{attribute 'GeneratedUsingTerminal: IODEVICETYPE_ETHERCATPROT'}
{attribute addProperty BoxType "IODEVICETYPE_ETHERCATPROT"}
{attribute addProperty Id "Beckhoff_EM2xxxBeckhoff_EM2xxx_23EB33C640Beckhoff_EM3xxxBeckhoff_EM3xxx_ABA3179978Beckhoff_EM7xxxBeckhoff_EM7xxx_110CC3B3681SyncUnitsSyncUnits_99E584AF18InputsInputs_25A0042B160OutputsOutputs_2397A10E106InfoDataInfoData_E68C61CD28"}
{attribute addProperty CRC "1180849743"}
{attribute addProperty Size "1111"}
TYPE EtherCAT_Master_EMxxxx_4662564F :
STRUCT
	{attribute addProperty Name "Beckhoff_EM2xxx"}
	{attribute addProperty PreviousPort "EtherCAT_Master_EMxxxx : Master"}
	Beckhoff_EM2xxx : Beckhoff_EM2xxx_23EB33C6;
	{attribute addProperty Name "Beckhoff_EM3xxx"}
	{attribute addProperty PreviousPort "Beckhoff EM2xxx : C"}
	Beckhoff_EM3xxx : Beckhoff_EM3xxx_ABA31799;
	{attribute addProperty Name "Beckhoff_EM7xxx"}
	{attribute addProperty PreviousPort "Beckhoff EM3xxx : C"}
	Beckhoff_EM7xxx : Beckhoff_EM7xxx_110CC3B3;
	{attribute addProperty Name "SyncUnits"}
	SyncUnits : SyncUnits_99E584AF;
	{attribute addProperty Name "Inputs"}
	Inputs : Inputs_25A0042B;
	{attribute addProperty Name "Outputs"}
	Outputs : Outputs_2397A10E;
	{attribute addProperty Name "InfoData"}
	InfoData : InfoData_E68C61CD;
END_STRUCT
END_TYPE

(* stored: Version 1.2.0.0, ProductVersion 3.1.4024.9
   DUT EtherCAT_Master_EMxxxx_4662564F: Id {e7be7e56-120a-45e1-ac15-50a80117e3af} *)
